(* Logix 5000 project; controller TF6280_CIP_Example 1769-L16ER-BB1B rev 32.11; software revision 32.00 *)

TASK MainTask (continuous, watchdog 500 ms) : MainProgram

MODULES
   Local : 1769-L16ER-BB1B (PointIO 0, rev 32.11)
      C6032 : vendor 108 type 12 code 6280 (Ethernet 192.168.40.111, rev 3.1, StandardDataDriven RPI 10 ms)
      Discrete_IO : Embedded (PointIO 1, rev 32.11, Output RPI 20 ms)
END_MODULES

VAR_GLOBAL   (* controller tags *)
   bGet : BOOL;   // Boolean trigger to Get attributes from Beckhoff
   bSet : BOOL;   // Boolean trigger to Set attributes at Beckhoff
   GetMsg : MESSAGE;   // Get message structure
        MessageParameters(ServiceCode := 16#000e, DestinationTag := RxData[0], ...)
   iAttriubuteSelect : INT := 1;   // A value from 1-3 to select the attribute message on Beckhoff side
   iCase : INT;   // Case statement variable
   iGet : INT;   // How many times the Get command has completed
   iLoop : INT := 81;   // Loop variable
   RxData : SINT[128];   // Rx Data Buffer
   SetMsg : MESSAGE;   // Set message structure
        MessageParameters(ServiceCode := 16#0010, LocalElement := TxData[0], ...)
   sGetAttribute : STRING;   // Last get message
   sSetAttribute : STRING := 'Hello Beckhoff';   // String to send on set
   TxData : SINT[128];   // Tx Data Buffer
END_VAR

PROGRAM MainProgram   (* main routine MainRoutine *)
VAR
   RxDataSize : DINT;
END_VAR

ROUTINE MainRoutine   (* structured text *)
   //Get Attribute Trigger
   IF bGet AND iCase = 0 AND iAttriubuteSelect <= 3 AND iAttriubuteSelect >= 1 THEN
       bGet:=0;
       iCase:=10 + iAttriubuteSelect;
   END_IF;
   
   //Set Attribute Trigger
   IF bSet AND iCase = 0 THEN
       bSet:=0;
       iCase:=40;
   END_IF;
   
   
   
   // Main Messaging Case Statement
   CASE iCase OF
   	11: //TestReadOnlyAttribute1
   	    GetMsg.Class:=16#1000;
   	    GetMsg.Instance:=16#01;
   	    GetMsg.Attribute:=16#01;
   	    iCase:=30;
   
   
   	12: //TestReadOnlyAttribute2
   	    GetMsg.Class:=16#1000;
   	    GetMsg.Instance:=16#01;
   	    GetMsg.Attribute:=16#02;
   	    iCase:=30;
   
   
   	23: //TestReadOnlyAttribute3
   	    GetMsg.Class:=16#1000;
   	    GetMsg.Instance:=16#01;
   	    GetMsg.Attribute:=16#03;
   	    iCase:=30;
   
   	30: //Get Attribue
   	    MSG(GetMsg);
   	    IF GetMsg.DN OR GetMsg.ER THEN
   			// Increment the successful counter
   	        iGet:=iGet+1;
   			// Prepare the string to display with only the character lenght
   			sGetAttribute.LEN := 22;
   			// Copy it to a string
   			SIZE(RxData,0, RxDataSize);
   			COP(RxData[0], sGetAttribute.DATA[0], RxDataSize);
   			// Return to wait state
   	        iCase:=0;
   	    END_IF;
   
   	40: // Set Attribute
   		// Copy the string into the TxData array
   		COP(sSetAttribute.DATA[0], TxData[0], 80);
   		// Send the message
   		MSG(SetMsg);
   		IF SetMsg.DN OR SetMsg.ER THEN
   			// Clear out the data buffer for next message
   			FOR iLoop := 0 TO 80 DO
   				TxData[iLoop] := 0;
   			END_FOR;
   			iCase := 0;
   		END_IF;
   END_CASE;
END_ROUTINE
END_PROGRAM
